INTERFACE I_StackLight_1

PROPERTY MyInput : BOOL
GET
END_GET
SET
END_SET
END_PROPERTY

PROPERTY MyOutput : E_PMLState
GET
END_GET
SET
END_SET
END_PROPERTY

END_INTERFACE

(* stored: Version 1.1.0.1
   Itf I_StackLight_1: Id {5e10ab32-d765-450b-a459-d1627f19852a}
   Property MyInput: Id {92b68c4e-e8a3-4d62-b91c-f7c40800d1b3}
   Get Get: Id {c0a24b52-5905-4ed3-8921-293678988eb7}
   Set Set: Id {fb22be43-898c-4a98-b3c0-caa7fc542542}
   Property MyOutput: Id {830c2886-3bec-41c3-920a-e8a2fdb7e4d1}
   Get Get: Id {45605781-491b-48a9-afc1-2e29894701af}
   Set Set: Id {c8f83b8d-b100-4431-84f6-7bee2896e413} *)
